(* IEC 61131-3 sources: TSA-FMICS22/ahorn/test/file, 57 files *)

(* ---- call_recursion.st ---- *)
PROGRAM P
VAR_INPUT
    x : INT;
END_VAR
VAR_OUTPUT
    y : INT;
END_VAR
VAR
    z : INT;
    f : Fb1;
    g : Fb2;
END_VAR
    f(z:=x,c=>y);
    IF y > 1 THEN
        g(x:=x);
    ELSE
        g(x:=x,b=>y);
    END_IF;
END_PROGRAM

FUNCTION_BLOCK Fb1
VAR_INPUT
    x : INT;
    y : INT;
    z : INT;
END_VAR
VAR_OUTPUT
    a : INT;
    b : INT;
    c : INT;
END_VAR
VAR
    g : Fb2;
END_VAR;
    a := x + 1;
    g(x:=y,y:=z,a=>b);
    IF g.b > 0 THEN
        c := 0;
    ELSE
        c := b + a;
    END_IF;
END_FUNCTION_BLOCK

FUNCTION_BLOCK Fb2
VAR_INPUT
    x : INT;
    y : INT;
END_VAR
VAR
    g : Fb2;
END_VAR
VAR_OUTPUT
    a : INT;
    b : INT;
END_VAR
    a := x + y;
    b := 2 * a;
END_FUNCTION_BLOCK

(* ---- chc_call.st ---- *)
PROGRAM P
VAR
    x : BOOL;
    y : INT;
    z : Fb;
END_VAR
    z(x:=x,y=>y);
END_PROGRAM

FUNCTION_BLOCK Fb
VAR_INPUT
    x : BOOL;
END_VAR
VAR_OUTPUT
    y : INT;
END_VAR
    IF x THEN
        y := 10;
    ELSE
        y := 20;
    END_IF;
END_FUNCTION_BLOCK

(* ---- chc_call_in_call.st ---- *)
PROGRAM P
VAR
    x : BOOL;
    y : INT;
    z : Fb1;
END_VAR
    z(x:=x,y=>y);
END_PROGRAM

FUNCTION_BLOCK Fb1
VAR_INPUT
    x : BOOL;
END_VAR
VAR
    z : Fb2;
END_VAR
VAR_OUTPUT
    y : INT;
END_VAR
    IF x THEN
        y := 10;
    ELSE
        z(x:=TRUE,y=>y);
    END_IF;
END_FUNCTION_BLOCK

FUNCTION_BLOCK Fb2
VAR_INPUT
    x : BOOL;
END_VAR
VAR_OUTPUT
    y : INT;
END_VAR
    IF x THEN
        y := 50;
    ELSE
        y := 20;
    END_IF;
END_FUNCTION_BLOCK

(* ---- chc_lower_ir_small_example.st ---- *)
PROGRAM P
VAR
    x : BOOL;
    y : INT;
    z : Fb;
END_VAR
    IF x THEN
        IF x > 0 THEN
            y := 2;
        ELSE
            IF x > 10 THEN
                y := 14;
            ELSE
                z(x:=y);
            END_IF;
        END_IF;
    ELSE
        y := 30;
    END_IF;
END_PROGRAM

FUNCTION_BLOCK Fb
VAR_INPUT
    x : INT;
END_VAR
    x := x + 1;
END_FUNCTION_BLOCK

(* ---- ir_call.st ---- *)
PROGRAM P
VAR_INPUT
    x : INT;
END_VAR
VAR_OUTPUT
    y : INT;
END_VAR
VAR
    z : INT;
    f : Fb1;
    g : Fb2;
END_VAR
    f(z:=x,c=>y);
    IF y > 1 THEN
        g(x:=x);
    ELSE
        g(x:=x,b=>y);
    END_IF;
END_PROGRAM

FUNCTION_BLOCK Fb1
VAR_INPUT
    x : INT;
    y : INT;
    z : INT;
END_VAR
VAR_OUTPUT
    a : INT;
    b : INT;
    c : INT;
END_VAR
VAR
    g : Fb2;
END_VAR;
    a := x + 1;
    g(x:=y,y:=z,a=>b);
    IF g.b > 0 THEN
        c := 0;
    ELSE
        c := b + a;
    END_IF;
END_FUNCTION_BLOCK

FUNCTION_BLOCK Fb2
VAR_INPUT
    x : INT;
    y : INT;
END_VAR
VAR_OUTPUT
    a : INT;
    b : INT;
END_VAR
    a := x + y;
    b := 2 * a;
END_FUNCTION_BLOCK

(* ---- parse_in_order.st ---- *)
PROGRAM P
VAR_INPUT
    x : INT;
END_VAR
VAR_OUTPUT
    y : INT;
END_VAR
VAR
    z : INT;
    h : Fb3;
    f : Fb1;
    g : Fb2;
END_VAR
    f(z:=x,c=>y);
    IF y > 1 THEN
        g(x:=x);
    ELSE
        g(x:=x,b=>y);
    END_IF;
END_PROGRAM

FUNCTION_BLOCK Fb3
VAR_INPUT
    x : INT;
    y : INT;
    z : INT;
END_VAR
VAR_OUTPUT
    a : INT;
END_VAR
VAR
    f : Fb1;
END_VAR;
    a := x + 1;
    f(x:=y,y:=z,a=>a);
END_FUNCTION_BLOCK

FUNCTION_BLOCK Fb1
VAR_INPUT
    x : BOOL;
    y : INT;
    z : INT;
END_VAR
VAR_OUTPUT
    a : INT;
    b : INT;
    c : INT;
END_VAR
VAR
    g : Fb2;
END_VAR;
    a := x + 1;
    g(x:=y,y:=z,a=>b);
    IF g.b > 0 THEN
        c := 0;
    ELSE
        c := b + a;
    END_IF;
END_FUNCTION_BLOCK

FUNCTION_BLOCK Fb2
VAR_INPUT
    x : INT;
    y : INT;
END_VAR
VAR_OUTPUT
    a : INT;
    b : INT;
END_VAR
    a := x + y;
    b := 2 * a;
END_FUNCTION_BLOCK

(* ---- pdg_call.st ---- *)
PROGRAM P
VAR_INPUT
    activate : BOOL;
END_VAR
VAR
    k : FbB;
    j : FbC;
    b : BOOL;
    y : INT;
    z : INT;
END_VAR
    IF b THEN
        k(q:=b,h=>z);
        j(q:=b,h=>z);
    ELSE
        WHILE y > 0 DO
            j(q:=b,h=>z);
            k(q:=b,h=>z);
        END_WHILE;
    END_IF;
    b := TRUE;
END_PROGRAM

FUNCTION_BLOCK FbB
VAR_INPUT
    q : BOOL;
END_VAR
VAR_OUTPUT
    h : INT;
END_VAR
    IF q THEN
        h := 1;
    ELSE
        h := 2;
    END_IF;
END_FUNCTION_BLOCK

FUNCTION_BLOCK FbC
VAR_INPUT
    q : BOOL;
END_VAR
VAR_OUTPUT
    h : INT;
END_VAR
    IF q THEN
        h := 1;
    ELSE
        h := 2;
    END_IF;
END_FUNCTION_BLOCK

(* ---- sa_call.st ---- *)
PROGRAM P
VAR_INPUT
    activate : BOOL;
END_VAR
VAR
    k : Fb;
    b : BOOL;
    y : INT;
    z : INT;
END_VAR
    b := TRUE;
    k(q:=b,h=>z);
    IF NOT(activate) AND b THEN
        y := 0;
    ELSE
        IF activate OR NOT(b) THEN
            y := 1;
        ELSE
            y := 2;
        END_IF;
    END_IF;
END_PROGRAM

FUNCTION_BLOCK Fb
VAR_INPUT
    q : BOOL;
END_VAR
VAR_OUTPUT
    h : INT;
END_VAR
    IF q THEN
        h := 1;
    ELSE
        h := 2;
    END_IF;
END_FUNCTION_BLOCK

(* ---- sa_call_parameters.st ---- *)
PROGRAM P
VAR_INPUT
    activate : BOOL;
END_VAR
VAR
    k : Fb;
    b : BOOL;
    y : INT;
    z1 : INT;
    z2 : INT;
    z3 : INT;
    z4 : INT;
END_VAR
    b := TRUE;
    k(r:=b AND b AND b,t:=b,q:=b OR TRUE,s:=FALSE,j=>z3,h=>z1,k=>z4,i=>z2);
    IF NOT(activate) AND b THEN
        y := 0;
    ELSE
        IF activate OR NOT(b) THEN
            y := 1;
        ELSE
            y := 2;
        END_IF;
    END_IF;
END_PROGRAM

FUNCTION_BLOCK Fb
VAR_INPUT
    q : BOOL;
    r : BOOL;
    s : BOOL;
    t : BOOL;
END_VAR
VAR_OUTPUT
    h : INT;
    i : INT;
    j : INT;
    k : INT;
END_VAR
    IF q THEN
        h := 1;
        i := 1;
        j := 1;
        k := 1;
    ELSE
        h := 2;
        i := 2;
        j := 2;
        k := 2;
    END_IF;
END_FUNCTION_BLOCK

(* ---- sa_ton.st ---- *)
PROGRAM P
VAR
    x : INT;
    y : TIME;
    T_1 : TON;
END_VAR
    IF T_1.Q THEN
        x := 0;
    ELSE
        x := 1;
    END_IF;
    T_1(IN:=TRUE,PT:=y);
END_PROGRAM

FUNCTION_BLOCK TON
VAR_INPUT
  IN : BOOL;
  PT : TIME;
END_VAR
VAR
  running : BOOL;
END_VAR
VAR_TEMP
    timeout : BOOL;
END_VAR
VAR_OUTPUT
  Q : BOOL;
  ET : TIME;
END_VAR
  timeout := NONDETERMINISTIC_BOOL();
  IF NOT IN THEN
    Q := FALSE;
    running := FALSE;
  ELSIF NOT running AND NOT Q THEN
    running := TRUE;
  ELSIF running AND NOT Q THEN
    Q := timeout;
    running := NOT Q;
  END_IF;

  ET := NONDETERMINISTIC_TIME();
END_FUNCTION_BLOCK

(* ---- se_engine_if_in_callee.st ---- *)
PROGRAM P
VAR_INPUT
    x : INT;
END_VAR
VAR
    f : Fb;
END_VAR
VAR_OUTPUT
    y : BOOL;
END_VAR
    f(a:=x,b=>y);
END_PROGRAM

FUNCTION_BLOCK Fb
VAR_INPUT
    a : INT;
END_VAR
VAR_OUTPUT
    b : BOOL;
END_VAR
IF a > 32 THEN
    b := TRUE;
ELSE
    b := FALSE;
END_IF;
END_FUNCTION_BLOCK

(* ---- se_executor_call.st ---- *)
PROGRAM P
VAR_INPUT
    x : INT;
END_VAR
VAR
    f : Fb;
END_VAR
VAR_OUTPUT
    y : INT;
END_VAR
    f(a:=x,b=>y);
END_PROGRAM

FUNCTION_BLOCK Fb
VAR_INPUT
    a : INT;
END_VAR
VAR_OUTPUT
    b : INT;
END_VAR;
    IF a >= 32 THEN
        b := 64;
    ELSE
        b := 16;
    END_IF;
END_FUNCTION_BLOCK

(* ---- se_executor_call_local_path_constraints.st ---- *)
PROGRAM P
VAR_INPUT
    x : INT;
END_VAR
VAR
    f : Fb1;
END_VAR
VAR_OUTPUT
    y : INT;
END_VAR
    f(a:=x,b=>y);
END_PROGRAM

FUNCTION_BLOCK Fb1
VAR_INPUT
    a : INT;
END_VAR
VAR
    f : Fb2;
END_VAR
VAR_OUTPUT
    b : INT;
END_VAR;
    IF a >= 32 THEN
        f(c:=x,d=>b);
    ELSE
        b := 16;
    END_IF;
END_FUNCTION_BLOCK

FUNCTION_BLOCK Fb2
VAR_INPUT
    c : INT;
END_VAR
VAR_OUTPUT
    d : INT;
END_VAR;
    IF c >= 32 THEN
        d := 64;
    ELSE
        d := 16;
    END_IF;
END_FUNCTION_BLOCK

(* ---- se_executor_call_with_state.st ---- *)
PROGRAM P
VAR_INPUT
    x : INT;
END_VAR
VAR
    f : Fb;
END_VAR
VAR_OUTPUT
    y : INT;
END_VAR
    f(a:=x,c=>y);
END_PROGRAM

FUNCTION_BLOCK Fb
VAR_INPUT
    a : INT;
END_VAR
VAR
    b : INT;
END_VAR
VAR_OUTPUT
    c : INT;
END_VAR;
    IF a >= 32 THEN
        b := b + 1;
    ELSE
        b := b - 1;
    END_IF;
    c := b;
END_FUNCTION_BLOCK

(* ---- se_executor_hagedorn_problem.st ---- *)
Program P
VAR_INPUT
    i : INT;
END_VAR
VAR
    f : Fb1;
    x : INT;
END_VAR
VAR_OUTPUT
    o : INT;
END_VAR
    x := i;
    IF change(FALSE,TRUE) THEN
        f(a:=x,b=>x);
    END_IF;
    o := change(i,x);
END_PROGRAM

FUNCTION_BLOCK Fb1
VAR_INPUT
    a : INT;
END_VAR
VAR_OUTPUT
    b : INT;
END_VAR
    b := a * 2;
END_FUNCTION_BLOCK

(* ---- se_executor_subsequent_calls.st ---- *)
PROGRAM P
VAR_INPUT
    x : INT;
END_VAR
VAR
    f : Fb;
END_VAR
VAR_OUTPUT
    y : INT;
END_VAR
    f(a:=x,b=>y);
    f(a:=x,b=>y);
END_PROGRAM

FUNCTION_BLOCK Fb
VAR_INPUT
    a : INT;
END_VAR
VAR_OUTPUT
    b : INT;
END_VAR;
    IF a >= 32 THEN
        b := 64;
    ELSE
        b := 16;
    END_IF;
END_FUNCTION_BLOCK

(* ---- chc_add.st ---- *)
PROGRAM P
VAR
    x : INT;
END_VAR
    x := x + 1;
END_PROGRAM

(* ---- chc_cycle_semantics.st ---- *)
PROGRAM P
VAR
    x : INT;
    y : INT;
END_VAR
    x := x + 1;
    IF x > 10 THEN
        y := 1;
    ELSE
        y := 0;
    END_IF;
END_PROGRAM

(* ---- chc_if.st ---- *)
PROGRAM P
VAR
    x : BOOL;
    y : INT;
END_VAR
    IF x THEN
        y := 1;
    ELSE
        y := 2;
    END_IF;
END_PROGRAM

(* ---- chc_lower_ir.st ---- *)
PROGRAM P
VAR
    x : BOOL;
    y : INT;
END_VAR
    IF x THEN
        y := 1;
    ELSE
        IF x THEN
            y := 2;
        ELSE
            y := 3;
        END_IF;
    END_IF;
END_PROGRAM

(* ---- chc_lower_ir_base_case_2.st ---- *)
PROGRAM P
VAR
    x : BOOL;
    y : INT;
END_VAR
    IF x THEN
        y := 1;
    END_IF;
END_PROGRAM

(* ---- chc_lower_ir_base_case_3.st ---- *)
PROGRAM P
VAR
    x : BOOL;
    y : INT;
END_VAR
    IF x THEN

    ELSE
        y := 1;
    END_IF;
END_PROGRAM

(* ---- chc_sub.st ---- *)
PROGRAM P
VAR
    x : INT;
END_VAR
    x := x - 1;
END_PROGRAM

(* ---- compiler_if.st ---- *)
PROGRAM P
VAR
    x : BOOL;
    y : INT;
END_VAR
    IF x > 0 THEN
        y := change(1,1);
    ELSE
        y := 2;
    END_IF;
END_PROGRAM

(* ---- compiler_if_else_if.st ---- *)
PROGRAM P
VAR
    x : BOOL;
    y : INT;
END_VAR
    IF x > 0 THEN
        y := 1;
    ELSIF x > 1 THEN
        y := 2;
    ELSE
        y := 3;
    END_IF;
END_PROGRAM

(* ---- ir_case.st ---- *)
PROGRAM P
VAR_INPUT
    x : INT;
END_VAR
VAR_OUTPUT
    code : WORD := 16#0000;
    result : WORD;
END_VAR
    (* Mismatch on purpose. Only first case should be reachable *)
    CASE code OF
    16#0000:
        code := 16#0001;
    16#0001:
        code := 16#0002;
    16#0002:
        code := 16#0003;
    16#0003:
        code := 16#0004;
    16#0004:
        code := 16#0000;
    END_CASE;

    result := code;
END_PROGRAM

(* ---- ir_empty_if.st ---- *)
PROGRAM P
VAR
    x : BOOL;
    y : INT;
END_VAR
    IF x > 0 THEN
    ELSE
    END_IF;
END_PROGRAM

(* ---- ir_empty_if_else_if_else.st ---- *)
PROGRAM P
VAR
    x : BOOL;
    y : INT;
END_VAR
    IF x > 0 THEN
    ELSIF x > 1 THEN
        y := 1;
    ELSE
        y := 2;
    END_IF;
END_PROGRAM

(* ---- ir_empty_if_empty_else_if_else.st ---- *)
PROGRAM P
VAR
    x : BOOL;
    y : INT;
END_VAR
    IF x > 0 THEN
    ELSIF x > 1 THEN
    ELSE
        y := 2;
    END_IF;
END_PROGRAM

(* ---- ir_enum.st ---- *)
TYPE
    Magazin_states_t : (Green_Lamp , Init , Interstep , Magazin_Init , Magazin_Init_2 , Slider_Move_Back , Start_Magazin , Step0 , Step1 , convey);
END_TYPE

PROGRAM P
VAR
    State : Magazin_states_t := Green_Lamp;
    x : INT;
END_VAR
    CASE State OF
    Green_Lamp:
        x := 1;
    Init:
        x := x + 1;
    Interstep:
        x := 2;
    Magazin_Init,
    Magazin_Init_2,
    Slider_Move_Back:
        x := 3;
    Start_Magazin,
    Step0:
        x := 4;
    Step1:
        x := 5;
    convey:
        x := 6;
    END_CASE;
END_PROGRAM

(* ---- ir_if.st ---- *)
PROGRAM P
VAR
    x : BOOL := TRUE;
    y : INT := 0;
END_VAR
    IF x > 0 THEN
        y := 1;
    ELSE
        y := 2;
    END_IF;
END_PROGRAM

(* ---- ir_if_change.st ---- *)
PROGRAM P
VAR
    x : BOOL;
    y : INT;
END_VAR
    IF x > 0 THEN
        y := change(1,2);
    ELSE
        y := 2;
    END_IF;
END_PROGRAM

(* ---- ir_if_else_if.st ---- *)
PROGRAM P
VAR
    x : BOOL;
    y : INT;
END_VAR
    IF x > 0 THEN
        y := 1;
    ELSIF x > 1 THEN
        y := 2;
        IF x > 5 THEN
            y := 5;
        ELSIF x > 40 THEN
            y := 20;
        ELSIF x > 10 THEN
            IF x > 10 THEN

            ELSIF x > 1 THEN
                y := 1;
            ELSE

            END_IF;
        ELSE
            y := 1;
        END_IF;
    ELSE
        IF x > 2 THEN
            y := 3;
        ELSE
            y := 4;
        END_IF;
    END_IF;
END_PROGRAM

(* ---- ir_if_empty_else.st ---- *)
PROGRAM P
VAR
    x : BOOL;
    y : INT;
END_VAR
    IF x > 0 THEN
        y := 2;
    ELSE
    END_IF;
END_PROGRAM

(* ---- ir_if_empty_else_if_else.st ---- *)
PROGRAM P
VAR
    x : BOOL;
    y : INT;
END_VAR
    IF x > 0 THEN
        y := 1;
    ELSIF x > 1 THEN

    ELSE
        y := 2;
    END_IF;
END_PROGRAM

(* ---- ir_if_empty_then.st ---- *)
PROGRAM P
VAR
    x : BOOL;
    y : INT;
END_VAR
    IF x > 0 THEN

    ELSE
        y := 2;
    END_IF;
END_PROGRAM

(* ---- ir_if_numeral.st ---- *)
PROGRAM P
VAR
    x : BOOL := TRUE;
    y : INT := 0;
END_VAR
    x := 1;
    IF x + 10 > 0 THEN
        y := 1;
    ELSE
        y := 2;
    END_IF;
END_PROGRAM

(* ---- ir_while.st ---- *)
PROGRAM P
VAR_INPUT
    i : INT;
END_VAR
VAR
    x : INT;
    z : INT;
END_VAR
    WHILE i > 0 DO
        IF x = 1 THEN
            z := 0;
        ELSE
            z := 1;
        END_IF;
        i := i - 1;
   END_WHILE;
END_PROGRAM

(* ---- pdg_example.st ---- *)
PROGRAM P
VAR_INPUT
    n_in : INT;
END_VAR
VAR
    n : INT;
    i : INT;
    sum : INT;
    prod : INT;
END_VAR
VAR_OUTPUT
    sum_out : INT;
    prod_out : INT;
END_VAR;
    n := n_input;
    i := 1;
    sum := 0;
    prod := 0;
    WHILE i <= n DO
        sum := sum + i;
        prod := prod * i;
        i := i + 1;
    END_WHILE;
    sum_out := sum;
    prod_out := prod;
END_PROGRAM

(* ---- sa_enum.st ---- *)
TYPE
    Magazin_states_t : (Green_Lamp , Init , Interstep , Magazin_Init , Magazin_Init_2 , Slider_Move_Back , Start_Magazin , Step0 , Step1 , convey);
END_TYPE

PROGRAM P
VAR
    x : INT;
    State : Magazin_states_t;
END_VAR
State := Magazin_states_t#Interstep;
CASE State OF
    Magazin_states_t#Green_Lamp:
        x := 0;

    Magazin_states_t#Init:
        x := 1;

    Magazin_states_t#Interstep:
        x := 2;

    Magazin_Init:
        x := 3;

    Magazin_Init_2:
        x := 4;

    Slider_Move_Back:
        x := 5;

    Start_Magazin:
        x := 6;

    Step0:
        x := 7;

    Step1:
        x := 8;

    convey:
        x := 9;
END_CASE;
END_PROGRAM

(* ---- sa_if_negation.st ---- *)
PROGRAM P
VAR_INPUT
    activate : BOOL;
END_VAR
VAR
    b : BOOL;
    y : INT;
END_VAR
    b := TRUE;
    IF NOT(activate) AND b THEN
        y := 0;
    ELSE
        IF activate OR NOT(b) THEN
            y := 1;
        ELSE
            y := 2;
        END_IF;
    END_IF;
END_PROGRAM

(* ---- sa_or.st ---- *)
PROGRAM P
VAR_INPUT
    Activate       : BOOL := FALSE;
END_VAR
VAR
    Ready          : BOOL := FALSE;
    S_TwoHandOut   : BOOL := FALSE;
    DiagCode       : WORD := 16#0;
END_VAR
IF NOT Activate THEN
 DiagCode := 16#0000;
ELSE
 CASE DiagCode OF
 16#0000:
     IF Activate THEN
          DiagCode := 16#8001;
     END_IF;
 END_CASE;
END_IF;

CASE DiagCode OF
16#0000:
  Ready := FALSE;
  S_TwoHandOut := FALSE;
16#8000:
  Ready := TRUE;
  S_TwoHandOut := TRUE;
16#8001:
  Ready := TRUE;
  S_TwoHandOut := FALSE;
END_CASE;
END_PROGRAM

(* ---- se_engine_if.st ---- *)
PROGRAM P
VAR_INPUT
    x : INT;
END_VAR
VAR
    y : BOOL;
END_VAR
IF x >= 32 THEN
    y := TRUE;
ELSE
    y := FALSE;
END_IF;
END_PROGRAM

(* ---- se_engine_nested_ifs.st ---- *)
PROGRAM P
VAR_INPUT
    x : INT;
END_VAR
VAR
    y : BOOL;
END_VAR
IF x > 32 THEN
    y := TRUE;
    IF x > 64 THEN
        y := FALSE;
    ELSE
        y := TRUE;
    END_IF;
ELSE
    y := FALSE;
    IF x < 16 THEN
        y := TRUE;
    ELSE
        y := FALSE;
    END_IF;
END_IF;
END_PROGRAM

(* ---- se_executor_change.st ---- *)
PROGRAM P
VAR
    x : INT;
    y : BOOL;
    z : BOOL;
END_VAR
    x := -1;
    y := change(TRUE, FALSE);
    z := NOT(y);
    x := z - y;
END_PROGRAM

(* ---- se_executor_concrete_assignments.st ---- *)
PROGRAM P
VAR
    x : INT;
    y : INT;
    z : INT;
END_VAR
    x := 1;
    y := 2;
    z := x + y;
    x := z - y;
END_PROGRAM

(* ---- se_executor_if.st ---- *)
PROGRAM P
VAR
    x : INT;
    y : INT;
END_VAR
    IF x >= 32 THEN
        y := 10;
    ELSE
        y := 20;
    END_IF;
END_PROGRAM

(* ---- se_executor_if_merge.st ---- *)
PROGRAM P
VAR_INPUT
    x : INT;
END_VAR
VAR
    y : INT;
END_VAR
    IF x >= 32 THEN
        y := 10;
    ELSE
        y := 20;
    END_IF;
END_PROGRAM

(* ---- se_executor_if_merge_different_versions.st ---- *)
PROGRAM P
VAR_INPUT
    a : INT;
END_VAR
VAR
    b : INT;
    c : INT;
    d : INT;
    e : INT;
    f : INT;
END_VAR
    a := a;
    f := a;
    c := f + b;
    IF c >= 32 THEN
        d := b + 1;
        b := a;
    ELSE
        d := b + e;
        e := c + 1;
    END_IF;
END_PROGRAM

(* ---- se_executor_if_merge_truly_symbolic_assignments.st ---- *)
PROGRAM P
VAR_INPUT
    x : INT;
END_VAR
VAR
    y : INT := 1;
    z : INT := 2;
END_VAR
    IF x >= 32 THEN
        x := x + y;
        y := x + z;
        z := y + 1;
        x := x + z;
        y := x;
    ELSE
        x := x + x;
        z := y + z;
        y := z + 4;
        x := y + z;
        y := x + 1;
        x := y + 1;
        y := y + 1;
        z := z + 2;
        z := z + z;
        x := z + 1;
    END_IF;
END_PROGRAM

(* ---- se_executor_input_assignments.st ---- *)
PROGRAM P
VAR_INPUT
    x : INT;
    y : INT;
END_VAR
VAR
    z : INT;
END_VAR
    z := x + y;
END_PROGRAM

(* ---- se_executor_symbolic_assignments.st ---- *)
PROGRAM P
VAR
    x : INT;
    y : INT := 5;
    z : INT := 3;
END_VAR
    x := x + 1;
    y := x + y - z;
    z := x + y;
    x := z - y;
END_PROGRAM

(* ---- se_executor_unary.st ---- *)
PROGRAM P
VAR
    x : INT;
    y : BOOL;
    z : BOOL;
END_VAR
    x := -1;
    y := TRUE;
    z := NOT(y);
    x := z - y;
END_PROGRAM

(* ---- se_executor_while.st ---- *)
PROGRAM P
VAR
    y : INT := 0;
END_VAR
    WHILE y < 16 DO
        y := y + 1;
    END_WHILE;
END_PROGRAM

(* ---- ssa_00.st ---- *)
PROGRAM P
VAR
    a : INT;
    b : INT;
    c : INT;
    d : INT;
END_VAR
    a := 42;
    b := a;
    c := a + b;
    a := c + 23;
    c := a + d;
END_PROGRAM

(* ---- ssa_tac_00.st ---- *)
PROGRAM P
VAR
    a : INT;
    b : INT;
    c : INT;
    d : INT;
END_VAR
    a := 42;
    b := a;
    c := a + b + b + a;
    a := c + 23 + a;
    IF a + b + c > 0 THEN
        a := 12 + 13 + 14 + 15;
    ELSE
        a := 2;
    END_IF;
    IF a >= 1 THEN
        b := b * b * b;
    END_IF;
END_PROGRAM

(* ---- ssa_wikipedia.st ---- *)
PROGRAM P
VAR
    w : INT;
    x : INT;
    y : INT;
    z : INT;
END_VAR
    x := 5;
    x := x - 3;
    IF x < 3 THEN
        y := x * 2;
        w := y;
    ELSE
        y := x - 3;
    END_IF;
    w := x - y;
    z := x + y;
END_PROGRAM
